// Mitsubishi GX Developer project: PLC_PCO520L2   PLC: Q06UDEH

PROGRAM CONFIG
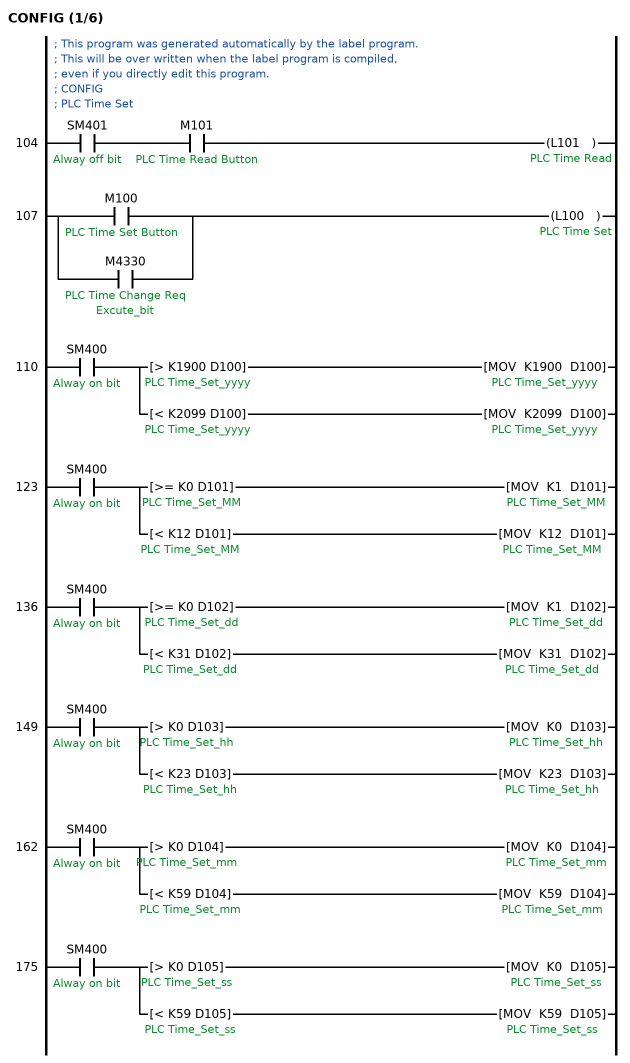
; This program was generated automatically by the label program.
; This will be over written when the label program is compiled,
; even if you directly edit this program.
; CONFIG
; 
; PLC Time Set
104   LD      SM401  ; Alway off bit
      AND     M101  ; PLC Time Read Button
      OUT     L101  ; PLC Time Read
107   LD      M100  ; PLC Time Set Button
      OR      M4330  ; PLC Time Change Req Excute_bit
      OUT     L100  ; PLC Time Set
110   LD      SM400  ; Alway on bit
      MPS
      AND>    K1900 D100  ; PLC Time_Set_yyyy
      MOV     K1900 D100
      MPP
      AND<    K2099 D100  ; PLC Time_Set_yyyy
      MOV     K2099 D100
123   LD      SM400  ; Alway on bit
      MPS
      AND>=   K0 D101  ; PLC Time_Set_MM
      MOV     K1 D101
      MPP
      AND<    K12 D101  ; PLC Time_Set_MM
      MOV     K12 D101
136   LD      SM400  ; Alway on bit
      MPS
      AND>=   K0 D102  ; PLC Time_Set_dd
      MOV     K1 D102
      MPP
      AND<    K31 D102  ; PLC Time_Set_dd
      MOV     K31 D102
149   LD      SM400  ; Alway on bit
      MPS
      AND>    K0 D103  ; PLC Time_Set_hh
      MOV     K0 D103
      MPP
      AND<    K23 D103  ; PLC Time_Set_hh
      MOV     K23 D103
162   LD      SM400  ; Alway on bit
      MPS
      AND>    K0 D104  ; PLC Time_Set_mm
      MOV     K0 D104
      MPP
      AND<    K59 D104  ; PLC Time_Set_mm
      MOV     K59 D104
175   LD      SM400  ; Alway on bit
      MPS
      AND>    K0 D105  ; PLC Time_Set_ss
      MOV     K0 D105
      MPP
      AND<    K59 D105  ; PLC Time_Set_ss
      MOV     K59 D105
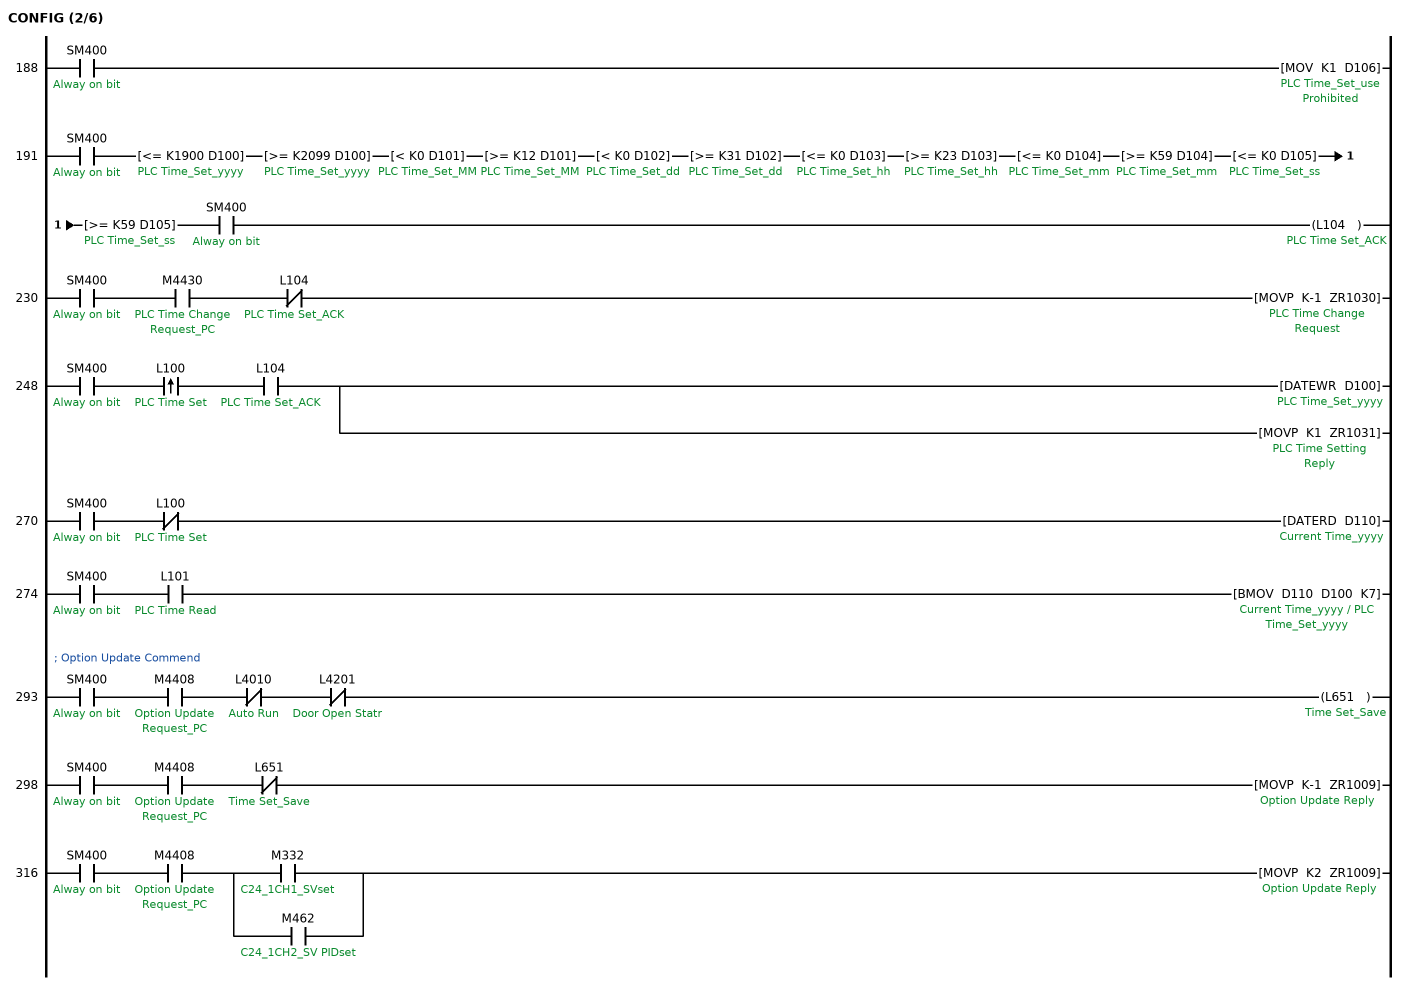
188   LD      SM400  ; Alway on bit
      MOV     K1 D106  ; PLC Time_Set_use Prohibited
191   LD      SM400  ; Alway on bit
      AND<=   K1900 D100  ; PLC Time_Set_yyyy
      AND>=   K2099 D100  ; PLC Time_Set_yyyy
      AND<    K0 D101  ; PLC Time_Set_MM
      AND>=   K12 D101  ; PLC Time_Set_MM
      AND<    K0 D102  ; PLC Time_Set_dd
      AND>=   K31 D102  ; PLC Time_Set_dd
      AND<=   K0 D103  ; PLC Time_Set_hh
      AND>=   K23 D103  ; PLC Time_Set_hh
      AND<=   K0 D104  ; PLC Time_Set_mm
      AND>=   K59 D104  ; PLC Time_Set_mm
      AND<=   K0 D105  ; PLC Time_Set_ss
      AND>=   K59 D105  ; PLC Time_Set_ss
      AND     SM400  ; Alway on bit
      OUT     L104  ; PLC Time Set_ACK
230   LD      SM400  ; Alway on bit
      AND     M4430  ; PLC Time Change Request_PC
      ANI     L104  ; PLC Time Set_ACK
      MOVP    K-1 ZR1030  ; PLC Time Change Request
        [note] PLC Time Change NAK
248   LD      SM400  ; Alway on bit
      ANDP    L100  ; PLC Time Set
      AND     L104  ; PLC Time Set_ACK
      DATEWR  D100
      MOVP    K1 ZR1031  ; PLC Time Setting Reply
        [note] PLC Time Change Complete
270   LD      SM400  ; Alway on bit
      ANI     L100  ; PLC Time Set
      DATERD  D110  ; Current Time_yyyy
274   LD      SM400  ; Alway on bit
      AND     L101  ; PLC Time Read
      BMOV    D110 D100 K7
; Option Update Commend
293   LD      SM400  ; Alway on bit
      AND     M4408  ; Option Update Request_PC
      ANI     L4010  ; Auto Run
      ANI     L4201  ; Door Open Statr
      OUT     L651  ; Time Set_Save
298   LD      SM400  ; Alway on bit
      AND     M4408  ; Option Update Request_PC
      ANI     L651  ; Time Set_Save
      MOVP    K-1 ZR1009  ; Option Update Reply
        [note] Option Update  Fail
316   LD      SM400  ; Alway on bit
      AND     M4408  ; Option Update Request_PC
      LD      M332  ; C24_1CH1_SVset
      OR      M462  ; C24_1CH2_SV PIDset
      ANB
      MOVP    K2 ZR1009
        [note] Option Update  Inprogres
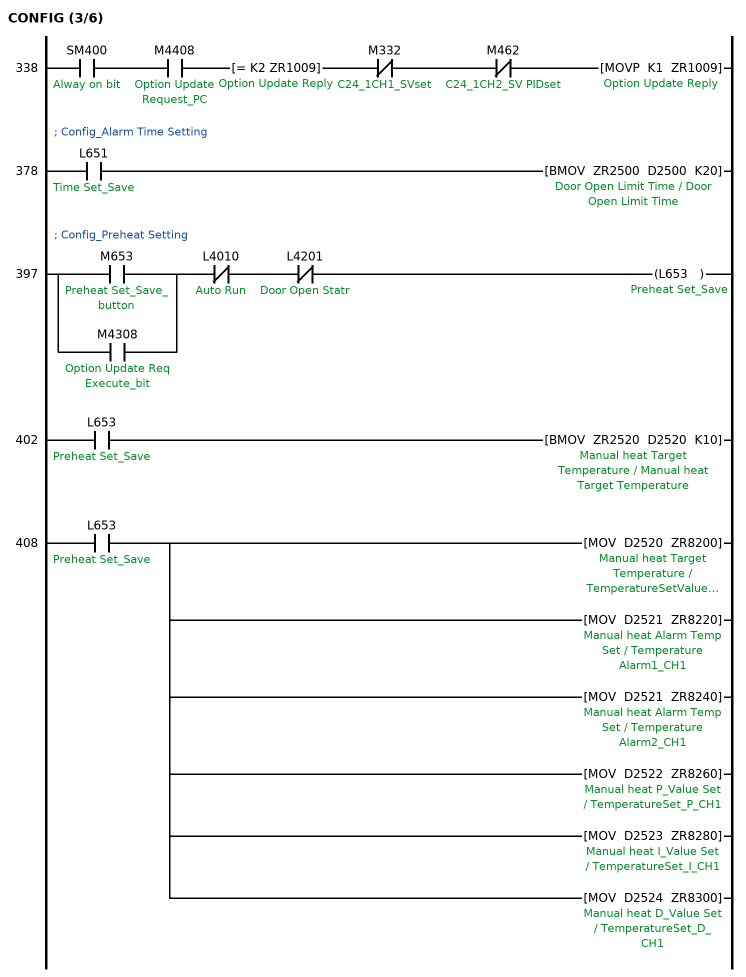
338   LD      SM400  ; Alway on bit
      AND     M4408  ; Option Update Request_PC
      AND=    K2 ZR1009  ; Option Update Reply
      ANI     M332  ; C24_1CH1_SVset
      ANI     M462  ; C24_1CH2_SV PIDset
      MOVP    K1 ZR1009
        [note] Option Update  Complete
; Config_Alarm Time Setting
378   LD      L651  ; Time Set_Save
      BMOV    ZR2500 D2500 K20  ; Door Open Limit Time / Door Open Limit Time
; Config_Preheat Setting
397   LD      M653  ; Preheat Set_Save_button
      OR      M4308  ; Option Update Req Execute_bit
      ANI     L4010  ; Auto Run
      ANI     L4201  ; Door Open Statr
      OUT     L653  ; Preheat Set_Save
402   LD      L653  ; Preheat Set_Save
      BMOV    ZR2520 D2520 K10  ; Manual heat Target Temperature / Manual heat Target Temperature
408   LD      L653  ; Preheat Set_Save
      MOV     D2520 ZR8200  ; TemperatureSetValue_CH1
      MOV     D2521 ZR8220  ; Manual heat Alarm Temp Set / TemperatureAlarm1_CH1
      MOV     D2521 ZR8240  ; TemperatureAlarm2_CH1
      MOV     D2522 ZR8260  ; Manual heat P_Value Set / TemperatureSet_P_CH1
      MOV     D2523 ZR8280  ; Manual heat I_Value Set / TemperatureSet_I_CH1
      MOV     D2524 ZR8300  ; Manual heat D_Value Set / TemperatureSet_D_CH1
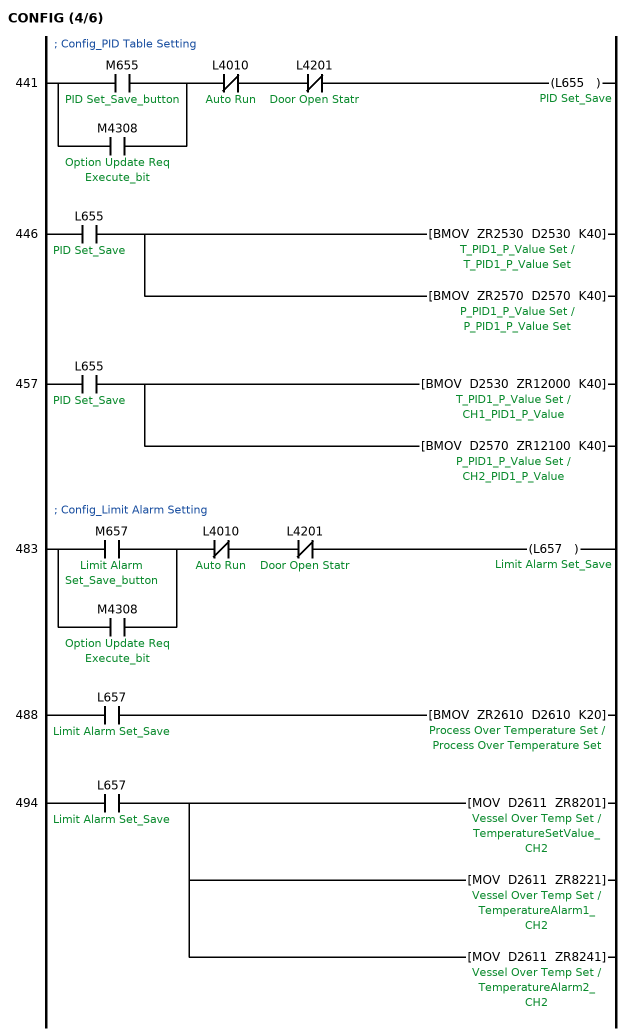
; Config_PID Table Setting
441   LD      M655  ; PID Set_Save_button
      OR      M4308  ; Option Update Req Execute_bit
      ANI     L4010  ; Auto Run
      ANI     L4201  ; Door Open Statr
      OUT     L655  ; PID Set_Save
446   LD      L655  ; PID Set_Save
      BMOV    ZR2530 D2530 K40  ; T_PID1_P_Value Set / T_PID1_P_Value Set
      BMOV    ZR2570 D2570 K40  ; P_PID1_P_Value Set / P_PID1_P_Value Set
457   LD      L655  ; PID Set_Save
      BMOV    D2530 ZR12000 K40  ; CH1_PID1_P_Value
      BMOV    D2570 ZR12100 K40  ; CH2_PID1_P_Value
; Config_Limit Alarm Setting
483   LD      M657  ; Limit Alarm Set_Save_button
      OR      M4308  ; Option Update Req Execute_bit
      ANI     L4010  ; Auto Run
      ANI     L4201  ; Door Open Statr
      OUT     L657  ; Limit Alarm Set_Save
488   LD      L657  ; Limit Alarm Set_Save
      BMOV    ZR2610 D2610 K20  ; Process Over Temperature Set / Process Over Temperature Set
494   LD      L657  ; Limit Alarm Set_Save
      MOV     D2611 ZR8201  ; Vessel Over Temp Set / TemperatureSetValue_CH2
      MOV     D2611 ZR8221  ; TemperatureAlarm1_CH2
      MOV     D2611 ZR8241  ; TemperatureAlarm2_CH2
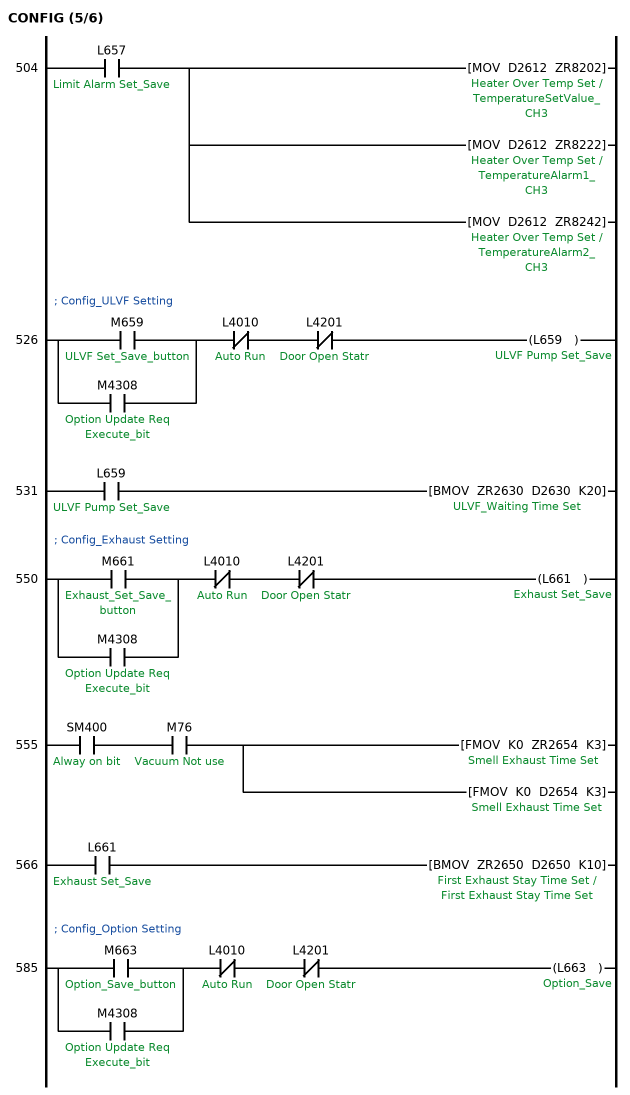
504   LD      L657  ; Limit Alarm Set_Save
      MOV     D2612 ZR8202  ; Heater Over Temp Set / TemperatureSetValue_CH3
      MOV     D2612 ZR8222  ; TemperatureAlarm1_CH3
      MOV     D2612 ZR8242  ; TemperatureAlarm2_CH3
; Config_ULVF Setting
526   LD      M659  ; ULVF Set_Save_button
      OR      M4308  ; Option Update Req Execute_bit
      ANI     L4010  ; Auto Run
      ANI     L4201  ; Door Open Statr
      OUT     L659  ; ULVF Pump Set_Save
531   LD      L659  ; ULVF Pump Set_Save
      BMOV    ZR2630 D2630 K20  ; ULVF_Waiting Time Set
; Config_Exhaust Setting
550   LD      M661  ; Exhaust_Set_Save_button
      OR      M4308  ; Option Update Req Execute_bit
      ANI     L4010  ; Auto Run
      ANI     L4201  ; Door Open Statr
      OUT     L661  ; Exhaust Set_Save
555   LD      SM400  ; Alway on bit
      AND     M76  ; Vacuum Not use
      FMOV    K0 ZR2654 K3  ; Smell Exhaust Time Set
      FMOV    K0 D2654 K3  ; Smell Exhaust Time Set
566   LD      L661  ; Exhaust Set_Save
      BMOV    ZR2650 D2650 K10  ; First Exhaust Stay Time Set / First Exhaust Stay Time Set
; Config_Option Setting
585   LD      M663  ; Option_Save_button
      OR      M4308  ; Option Update Req Execute_bit
      ANI     L4010  ; Auto Run
      ANI     L4201  ; Door Open Statr
      OUT     L663  ; Option_Save
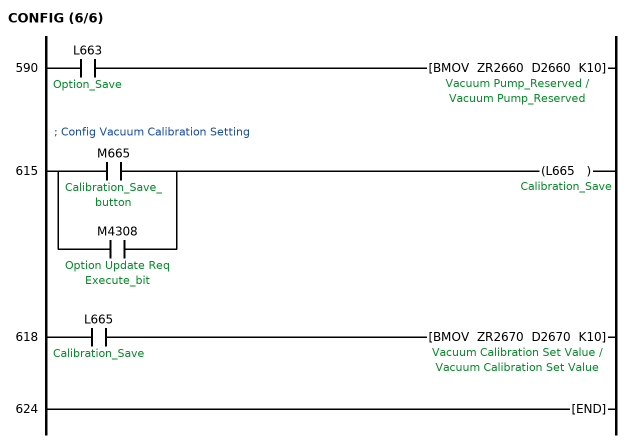
590   LD      L663  ; Option_Save
      BMOV    ZR2660 D2660 K10  ; Vacuum Pump_Reserved / Vacuum Pump_Reserved
; Config Vacuum Calibration Setting
615   LD      M665  ; Calibration_Save_button
      OR      M4308  ; Option Update Req Execute_bit
      OUT     L665  ; Calibration_Save
618   LD      L665  ; Calibration_Save
      BMOV    ZR2670 D2670 K10  ; Vacuum Calibration Set Value / Vacuum Calibration Set Value
624   END
END_PROGRAM
